// TIA Portal V20 export
TYPE "UDT_DefinicionDispositivo"
   STRUCT
      EventosDelJdT02 : Bool;
      ExisteSirena : Bool;
   END_STRUCT;
END_TYPE
